INTERFACE IFuseChannelBasic EXTENDS __SYSTEM.IQueryInterface

PROPERTY CoolDownLock  : bool
GET
END_GET
END_PROPERTY

PROPERTY CurrentLevelWarning  : bool
GET
END_GET
END_PROPERTY

PROPERTY Diag  : bool
GET
END_GET
END_PROPERTY

PROPERTY Enabled : bool
GET
END_GET
END_PROPERTY

PROPERTY Error  : bool
GET
END_GET
END_PROPERTY

PROPERTY HardwareProtection : bool
GET
END_GET
END_PROPERTY

METHOD ResetFuse : BOOL
END_METHOD

PROPERTY StateReset : bool
GET
END_GET
END_PROPERTY

PROPERTY StateSwitch : bool
GET
END_GET
END_PROPERTY

METHOD SwitchFuse : BOOL
END_METHOD

PROPERTY Tripped : bool
GET
END_GET
END_PROPERTY

PROPERTY TxPDOState  : bool
GET
END_GET
END_PROPERTY

END_INTERFACE

(* stored: Version 1.1.0.1, ProductVersion 3.1.4024.5
   Itf IFuseChannelBasic: Id {7103bcc3-8451-4f79-98e1-5e6cfa305d23}
   Property CoolDownLock: Id {b1d417c3-423e-44ef-b643-f33c47c7f09d}
   Get Get: Id {ca4851fb-648b-4448-b724-c6b9b7cbd7be}
   Property CurrentLevelWarning: Id {f07fc940-b0af-4df5-839e-5f41f6e4d6a3}
   Get Get: Id {24502174-5c12-4dfa-9708-8d3bab2b553c}
   Property Diag: Id {37b496c3-caff-4fff-a2fb-134a05867066}
   Get Get: Id {75103b0d-e69a-4e16-a310-32eb1390eb23}
   Property Enabled: Id {bd933298-6b1b-4d72-9f6c-9f804dfef166}
   Get Get: Id {d6d092c8-c845-4f4c-a197-e9315299834d}
   Property Error: Id {f2ed4433-d5dc-4cd4-a97a-dc8960d6bc38}
   Get Get: Id {8db2ef0e-d88e-4f8e-8a2a-2210b4600580}
   Property HardwareProtection: Id {b4d4d363-ceeb-42f4-86b5-082ed04486c9}
   Get Get: Id {361a1f32-bfe9-4e42-910b-fec9724e3076}
   Method ResetFuse: Id {b805691e-3c17-48c8-a026-8d60eb100362}
   Property StateReset: Id {2321444f-4a54-403c-8b72-7ffdf6603036}
   Get Get: Id {3f47ab45-5de3-4b35-a88e-36341d3a6c87}
   Property StateSwitch: Id {03496e87-1965-45a1-ac52-89d2428afae9}
   Get Get: Id {5323f810-fdb9-4ede-b3e5-f56b4fe78bdd}
   Method SwitchFuse: Id {3f803776-9e28-44ed-8210-828282c51c88}
   Property Tripped: Id {09cc707d-1ac5-4948-8856-5481eb82e5b5}
   Get Get: Id {fcddf3db-256f-4fe1-9a0b-20647e5453b5}
   Property TxPDOState: Id {ee9ec970-e0c3-4c4f-8ea6-ee09f32731cd}
   Get Get: Id {02836cb3-0772-4a0c-a66b-a6d8acf2c580} *)
